FUNCTION_BLOCK FB_RoomTemp

VAR
	_bInit					: BOOL;
	
	// fb:s
	_fbRoomTempControl		: FB_RoomTempControl;
	_fbCoolingControl		: FB_CoolingControl;
	
	_fbMotorCooling			: FB_MotorAbb880_malli;
	
	
END_VAR


_fbRoomTempControl();
_fbCoolingControl();

_fbMotorCooling();

//FB_Init is always available implicitly and it is used primarily for initialization.
//The return value is not evaluated. For a specific influence, you can also declare the
//methods explicitly and provide additional code there with the standard initialization
//code. You can evaluate the return value.
METHOD FB_Init: BOOL
VAR_INPUT
    bInitRetains: BOOL; // TRUE: the retain variables are initialized (reset warm / reset cold)
    bInCopyCode: BOOL;  // TRUE: the instance will be copied to the copy code afterward (online change)   
END_VAR
_bInit := TRUE;
END_METHOD

METHOD Init : BOOL
VAR_INPUT
END_VAR
IF _bInit THEN
	

_fbMotorCooling.Init( 	sName := 'Generaattorihuone jäähdytys moottori',
						refHmi := Motors.stMotors);

_fbRoomTempControl.Init(	refHmi		:= GVL.stRoomTemp,
							sName		:= 'Generaattori huone',
							iGenerator	:= GVL.fbGenerator);

_fbCoolingControl.Init(	refHmi		:= GVL.stCoolingControl,
						sName		:= 'Generaattori huoneen jäähdytys',
						iMotor		:= _fbMotorCooling,
						iRoomTemp	:= _fbRoomTempControl );


_bInit := FALSE;
END_IF
END_METHOD

END_FUNCTION_BLOCK

(* stored: Version 1.1.0.1
   POU FB_RoomTemp: Id {4e3d660a-5e64-4e2e-a474-66c0f3afef75}, SpecialFunc None
   Method FB_Init: Id {eba7c06a-cc1a-472b-a54e-5993b983ee8a}
   Method Init: Id {09c6c418-4d03-4883-b3d1-b789aa6be4c5} *)
